Fanuc KAREL source: kt00057.KL

PROGRAM KT00057
%NOLOCKGROUP
VAR
H1 : ARRAY[2] OF SHORT
I2:INTEGER
OUT:INTEGER
BEGIN
H1[1]=2
I2=3
OUT=(H1[1] - I2)
END KT00057
